FUNCTION_BLOCK RT_E_TRAIN (* Generation of a finite train of events *)
  (* Standard: 61499-2 *)
  (* Version 0.0, 2008-07-10, 4DIAC-IDE, 4DIAC-Consortium *)
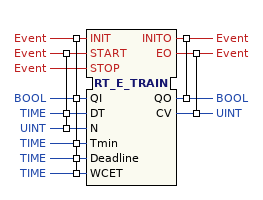
  EVENT_INPUT
    INIT WITH QI, Tmin, Deadline, WCET;
    START WITH DT, N;
    STOP;
  END_EVENT
  EVENT_OUTPUT
    INITO WITH QO;
    EO WITH CV; (* N events at period DT,starting at DT after START *)
  END_EVENT
  VAR_INPUT
    QI : BOOL;
    DT : TIME; (* Period between events *)
    N : UINT; (* Number of events to generate *)
    Tmin : TIME;
    Deadline : TIME;
    WCET : TIME;
  END_VAR
  VAR_OUTPUT
    QO : BOOL;
    CV : UINT; (* EO index(0 N-1) *)
  END_VAR
END_FUNCTION_BLOCK
